// TIA Portal V19 export
TYPE "IO Burkett Type 8691"
TITLE = Burkett_Type8691.rev2_Params
// DEVICEID : 2224898
//  VENDOR : Burkett
//  DATE: 27.12.2023 
// 
//  Comment : Burkett_Type8691.rev2_Params
   STRUCT
      V : Struct   // BURKETT_TYPE_8691 IO-LINK
         _IO : Struct   // Valve Control Interface
            IN : Struct
               Addr : Int;   // First Byte address of 4 byte address space
               Locate : Bool;   // Rapid Flash LED's
               Activate : Bool;   // Activate pilot valve
            END_STRUCT;
            OUT : Struct
               ValvePosition : Real;   // 0-100%
               Locate : Bool;   // Rapid Flash LED's
               NumarState : Byte;   // 0=diagPassive,1=diagActive,2=MaintenanceRequired,3=OutOfSpec,4=warn,5=error
               ValveMode : Byte;   // 0=Initialisation, 1=Normal Operation, 2=Teach function active, 3=SafePos active
               ValveOpened : Bool;
               ValveClosed : Bool;
               O_DI4 : Bool;   // Output signal status Pin 4
               O_DI2 : Bool;   // Output signal status Pin 2
               O_DA : Bool;   // Output device recognised
               O_DE : Bool;   // Output device error event has appeared
               O_PQ : Bool;   // Output port qualifer proces data valid
            END_STRUCT;
            IN_OUT : Struct
               HMI_CMD : Word;
               HMI_INFO : Word;
            END_STRUCT;
         END_STRUCT;
      END_STRUCT;
   END_STRUCT;
END_TYPE
